// TIA Portal V16 export
// export: Created 2022-11-01T21:54:10.0380842Z, ExportSetting WithDefaults, DisplayName Totally Integrated Automation Portal, DisplayVersion V16, DisplayName TIA Portal Version Control Interface, DisplayVersion V16, DisplayName TIA Portal Openness, DisplayVersion V16, DisplayName SINAMICS Startdrive Advanced, DisplayVersion V16, DisplayName SINAMICS Startdrive G130, G150, S120, S150, SINAMICS MV, S210, DisplayVersion V16, DisplayName SINAMICS Startdrive G110M, G120, G120C, G120D, G120P, DisplayVersion V16, DisplayName STEP 7 Professional, DisplayVersion V16, DisplayName STEP 7 Safety, DisplayVersion V16, DisplayName WinCC Professional, DisplayVersion V16
VAR_GLOBAL   // PLC tag table "AI C500"
   iTIR501 AT %IW1600 : Int;
   iTIR502 AT %IW1602 : Int;
   iTIR503 AT %IW1604 : Int;
   iTIR504 AT %IW1606 : Int;
   iTIR505 AT %IW1608 : Int;
   iTIR506 AT %IW1610 : Int;
   iTIR507 AT %IW1612 : Int;
   iTIR508 AT %IW1614 : Int;
   iTIR509 AT %IW1616 : Int;
   iTIR510 AT %IW1618 : Int;
   iTIR511 AT %IW1620 : Int;
   iTIR512 AT %IW1622 : Int;
   iTIR513 AT %IW1624 : Int;
   iTIR514 AT %IW1626 : Int;
   iTIR515 AT %IW1628 : Int;
   iTIR516 AT %IW1630 : Int;
   iTIR517 AT %IW1632 : Int;
   iTIR518 AT %IW1634 : Int;
   iTIR519 AT %IW1636 : Int;
   iTIR520 AT %IW1638 : Int;
   iTIR521 AT %IW1640 : Int;
   iTIR522 AT %IW1642 : Int;
   iTIR523 AT %IW1644 : Int;
   iTIR524 AT %IW1646 : Int;
   iTIR525 AT %IW1648 : Int;
   iTIR526 AT %IW1650 : Int;
   iTIR527 AT %IW1652 : Int;
   iTIR528 AT %IW1654 : Int;
   iPIR501 AT %IW1656 : Int;
   iPIR502 AT %IW1658 : Int;
   iPIR503 AT %IW1660 : Int;
   iPIR504 AT %IW1662 : Int;
   iPIR505 AT %IW1664 : Int;
   iPIR506 AT %IW1666 : Int;
   iPIR507 AT %IW1668 : Int;
   iPIR508 AT %IW1670 : Int;
   iPIR509 AT %IW1672 : Int;
   iPIR510 AT %IW1674 : Int;
   iPIR511 AT %IW1676 : Int;
   iLIR501 AT %IW1678 : Int;
   iLIR502 AT %IW1680 : Int;
   iLIR503 AT %IW1682 : Int;
   iLIR504 AT %IW1684 : Int;
   iLIR505 AT %IW1686 : Int;
   iLIR506 AT %IW1688 : Int;
   iLIR507 AT %IW1690 : Int;
   iLIR508 AT %IW1692 : Int;
   iLIR509 AT %IW1694 : Int;
   iLIR510 AT %IW1696 : Int;
   iLIR511 AT %IW1698 : Int;
   iLIR512 AT %IW1700 : Int;
   iLIR513 AT %IW1702 : Int;
   iLIR514 AT %IW1704 : Int;
   iLIR515 AT %IW1706 : Int;
   iLIR516 AT %IW1708 : Int;
   iLIR517 AT %IW1710 : Int;
   iLIR518 AT %IW1712 : Int;
   iLIR519 AT %IW1714 : Int;
   iLIR520 AT %IW1716 : Int;
   iLIR521 AT %IW1718 : Int;
   iLIR522 AT %IW1720 : Int;
   iFIR501 AT %IW1722 : Int;
   iFIR502 AT %IW1724 : Int;
   iFIR503 AT %IW1726 : Int;
   iFIR504 AT %IW1728 : Int;
   iFIR505 AT %IW1730 : Int;
   iFIR506 AT %IW1732 : Int;
   iFIR507 AT %IW1734 : Int;
   iFIR508 AT %IW1736 : Int;
   iFIR509 AT %IW1738 : Int;
   iFIR510 AT %IW1740 : Int;
   iFIR511 AT %IW1742 : Int;
   iFIR512 AT %IW1744 : Int;
   iFIR513 AT %IW1746 : Int;
   iFIR514 AT %IW1748 : Int;
   iFIR515 AT %IW1750 : Int;
   iFIR516 AT %IW1752 : Int;
   "iTIR514-1" AT %IW1754 : Int;
END_VAR
